// TIA Portal V20 export
DATA_BLOCK "IdentMvHmi"   // DB214
// stored: MemoryReserve 100
   VAR
      unitIdentMv : Array[1.."NO_OF_UNITS"] of "typeEMIdentMv";
   END_VAR
BEGIN
END_DATA_BLOCK
